// TIA Portal V20 export
// export: Created 2026-08-08T00:00:00.0000000Z, ExportSetting WithDefaults, DisplayName Totally Integrated Automation Portal, DisplayVersion V20, DisplayName TIA Portal Openness, DisplayVersion V20, DisplayName TIA Portal Version Control Interface, DisplayVersion V20, DisplayName STEP 7 Professional, DisplayVersion V20, DisplayName STEP 7 Safety, DisplayVersion V20, DisplayName WinCC Basic/Comfort/Advanced, DisplayVersion V20, DisplayName WinCC Professional, DisplayVersion V20, DisplayName WinCC Unified, DisplayVersion V20
TYPE "UDT_Valve_Config"
// Per-valve physical channel assignment. 0 = unassigned (valve runs on symbolic simulation). A nonzero value is an index into IO_Buffer_DB.DI[]/DQ[] - our own abstract channel numbering, translated to real hardware addresses in one place only (see FC_IoMapper).
// stored: IsFailsafeCompliant false
   STRUCT
      OpenFb_Channel : Int;
      ClosedFb_Channel : Int;
      Healthy_Channel : Int;
      LocalMode_Channel : Int;
      OpenCmd_Channel : Int;
      CloseCmd_Channel : Int;
   END_STRUCT;
END_TYPE
